{attribute 'qualified_only'}
{attribute 'strict'}
{attribute 'to_string'}
TYPE E_3002_2_Enable_manual_control : (
		Enable_control	:= 0,
		Disable_control := 1
	) UINT;
END_TYPE

(*
Used to enable manual control from this section:
	0 - Enable control
Navitrol will activate manual mode and sets WARNING_ETH_MANUAL_MODE. This section can be used to drive the AGV.
	1 - Disable control
Navitrol will ignore any controls from this section.
*)

(* stored: Version 1.1.0.1, ProductVersion 3.1.4026.17
   DUT E_3002_2_Enable_manual_control: Id {bf3ac82e-90d0-4903-868d-30605172a7e7} *)
